FUNCTION TryConvert_TIME_TO_ULINT : BOOL
VAR_INPUT
	in : TIME;
	out : REFERENCE TO ULINT;
END_VAR

out := TIME_TO_ULINT(in);
TryConvert_TIME_TO_ULINT := TRUE;

END_FUNCTION

(* stored: Version 1.1.0.1, ProductVersion 3.1.4024.12
   POU TryConvert_TIME_TO_ULINT: Id {f458a98c-211b-4bea-8fd9-021b3cf063c6}, SpecialFunc None *)
